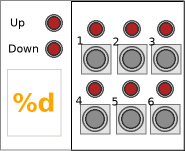
VISUALIZATION FloorControl  // 185x151
VAR_IN_OUT
	LED_Up	 		: BOOL;
	LED_Down		: BOOL;
	FloorNumber 	: INT;
	BtnLed	 		: ARRAY[1..6] OF BOOL;;
	Btn				: ARRAY[1..6] OF BOOL;
END_VAR
    RoundedRectangle (71,1 114x150)
    PushSwitch (81,44 30x30), variable: Btn[1], behaviour: TAP, style: Switch-PushSwitch-Gray
    Lamp1 (86,19 20x20), variable: BtnLed[1], style: Lamp-Lamp1-Red
    PushSwitch (117,44 30x30), variable: Btn[2], behaviour: TAP, style: Switch-PushSwitch-Gray
    Lamp1 (122,19 20x20), variable: BtnLed[2], style: Lamp-Lamp1-Red
    PushSwitch (151,44 30x30), variable: Btn[3], behaviour: TAP, style: Switch-PushSwitch-Gray
    Lamp1 (156,19 20x20), variable: BtnLed[3], style: Lamp-Lamp1-Red
    Lamp1 (44,13 20x20), variable: LED_Up, style: Lamp-Lamp1-Red
    Lamp1 (44,39 20x20), variable: LED_Down, style: Lamp-Lamp1-Red
    Label (70,31 20x20), "1"
    Label (106,32 20x20), "2"
    Label (142,32 20x20), "3"
    PushSwitch (80,104 30x30), variable: Btn[4], behaviour: TAP, style: Switch-PushSwitch-Gray
    Lamp1 (85,79 20x20), variable: BtnLed[4], style: Lamp-Lamp1-Red
    PushSwitch (116,104 30x30), variable: Btn[5], behaviour: TAP, style: Switch-PushSwitch-Gray
    Lamp1 (121,79 20x20), variable: BtnLed[5], style: Lamp-Lamp1-Red
    PushSwitch (150,104 30x30), variable: Btn[6], behaviour: TAP, style: Switch-PushSwitch-Gray
    Lamp1 (155,79 20x20), variable: BtnLed[6], style: Lamp-Lamp1-Red
    Label (69,91 20x20), "4"
    Label (105,92 20x20), "5"
    Label (141,92 20x20), "6"
    Label (7,13 36x20), "Up"
    Label (5,39 38x20), "Down"
    Textfield (7,69 54x67), "%d", text variable: FloorNumber
END_VISUALIZATION

(* stored: Version 1.1.0.1
   Visu FloorControl: Id {1eb610a1-ca66-459f-a3ba-606e2eba9c98} *)
